FUNCTION F_TzInfoBiasToTzStr : STRING
VAR_INPUT
	tzBias : DINT;
END_VAR
VAR
	UtcOffset : DINT;
END_VAR

UtcOffset := (0-tzBias) / 60;
IF UtcOffset > 0 AND UtcOffset < 10 THEN
	F_TzInfoBiasToTzStr := CONCAT(STR1:= 'UTC+0', STR2:= DINT_TO_STRING(UtcOffset));
ELSIF UtcOffset >= 10 AND UtcOffset <= 12 THEN
	F_TzInfoBiasToTzStr := CONCAT(STR1:= 'UTC+', STR2:= DINT_TO_STRING(UtcOffset));
ELSIF UtcOffset < 0 AND UtcOffset > -10 THEN
	F_TzInfoBiasToTzStr := CONCAT(STR1:= 'UTC-0', STR2:= DINT_TO_STRING(UtcOffset));
ELSIF UtcOffset <=10 AND UtcOffset >= -12 THEN
	F_TzInfoBiasToTzStr := CONCAT(STR1:= 'UTC-', STR2:= DINT_TO_STRING(UtcOffset));
ELSIF UtcOffset = 0 THEN
	F_TzInfoBiasToTzStr := 'UTC';
END_IF

END_FUNCTION

(* stored: Version 1.1.0.1, ProductVersion 3.1.4024.12
   POU F_TzInfoBiasToTzStr: Id {874d6c6f-5261-496a-aa14-1bc6118e7be6}, SpecialFunc None *)
